ADAPTER AQ (* unidirectional Adapter Interface for 1 Event and 1 Byte (containing 2 bits) *)
  (* Standard: 61499-1; Description: Copyright (c) 2026 Meisterschulen am Ostbahnhof SPDX-License-Identifier: EPL-2.0 *)
  (* Version 1.0, 2026-05-16, Franz Höpfinger, Meisterschulen am Ostbahnhof, Initial Version *)
  PACKAGE adapter::types::unidirectional;
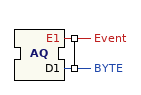
  EVENT_OUTPUT
    E1 WITH D1; (* Indication (or Request) Event from Plug *)
  END_EVENT
  VAR_OUTPUT
    D1 : BYTE; (* Indication (or Request) Data from Plug (2 bits) *)
  END_VAR
END_ADAPTER
